FUNCTION TryConvert_DINT_TO_WORD : BOOL
VAR_INPUT
	in : DINT;
	out : REFERENCE TO WORD;
END_VAR

IF in > DatatypeLimits.MAX_VALUE_OF_DINT_WHICH_CAN_BE_HELD_IN_A_WORD THEN
	RETURN;
END_IF

IF in < DatatypeLimits.MIN_VALUE_OF_DINT_WHICH_CAN_BE_HELD_IN_A_WORD THEN
	RETURN;
END_IF

out := DINT_TO_WORD(in);
TryConvert_DINT_TO_WORD := TRUE;

END_FUNCTION

(* stored: Version 1.1.0.1, ProductVersion 3.1.4024.12
   POU TryConvert_DINT_TO_WORD: Id {48cf2f57-700f-47aa-b1f7-7dffd7cdaaea}, SpecialFunc None *)
